Universal Robots PolyScope program: tip_test.urp

Program tip_test (installation=default directory=/programs createdIn=5.14.5 lastSavedIn=5.14.5 robotSerialNumber=20236801216)
Calibrated DH parameters: a=[-0.000021, -0.748897, -0.28186, -0.00004, -0.000055, 0]; d=[0.236225, -424.082933, -1564.66872, 1988.95162, 0.159094, 0.153873]; alpha=[1.570844, 0.001002, 0.000337, 1.571488, -1.569996, 0]; deltaTheta=[0, -0.516316, 5.626292, 1.173211, 0.000001, 0]
InitVariablesNode
Robot Program (runOnlyOnce=true)
  SafeHome (positionOptionType=SPEED_AND_ACCELERATION speed=1.047198 acceleration=1.396263 nextMotionTime=2)
  Set NoAction tcp=pretend_w_top
  MoveJ speed 60 deg/s, acceleration 80 deg/s^2 (useActiveTCP=true) feature=Base
    Waypoint Waypoint_2: TCP in base x=-2.094 y=-610.461 z=2075.593 mm, rx=-0.0011 ry=-2.2184 rz=2.2234 rad; joints [-0.001, -90.001, 0, -89.999, 0, 0.001] deg; TCP offset x=1.57 y=-90.08 z=257.67 mm, rx=0 ry=0 rz=0 rad
  MoveJ speed 200 deg/s, acceleration 200 deg/s^2 (useActiveTCP=true) feature=Base
    Waypoint Waypoint_1: TCP in base x=-1564.474 y=1111.87 z=503.05 mm, rx=1.8628 ry=0.7771 rz=-1.9631 rad; joints [-53.946, -7.314, -2.058, -90, 0, 0] deg
    Waypoint Waypoint_2: TCP in base x=-2.094 y=-610.461 z=2075.593 mm, rx=-0.0011 ry=-2.2184 rz=2.2234 rad; joints [-0.001, -90.001, 0, -89.999, 0, 0.001] deg
  SafeHome (positionOptionType=SPEED_AND_ACCELERATION speed=1.047198 acceleration=1.396263 nextMotionTime=2)
